PROGRAM Light
VAR
	Counter: int;
END_VAR

Counter := Counter +22;

END_PROGRAM

(* stored: Version 1.1.0.1, ProductVersion 3.1.4024.12
   POU Light: Id {be8ae8b6-ba5a-4031-acf9-6c804135e679}, SpecialFunc None *)
